(* Logix 5000 project; controller R5_CSS vendor 1 type 14 code 74 rev 19.11; software revision 19.01; part 4 of 20 *)
(* tags used below, declared in another part *)
   AlarmMaster : DINT;
   Coal_Tank_Heel_Inches : REAL;
   Coal_Tank_Height_Inches : REAL;
   FC101 : FLOW_CONTROL;   // QUENCH BASIN FLOW TRANSMITTER CONTROL
   FC108 : FLOW_CONTROL;   // QUENCH FEED FLOW TRANSMITTER
   FC140A : FLOW_CONTROL;   // QUENCH TOWER UPPER SPRAY FLOW CONTROL
   FC140B : FLOW_CONTROL;   // QUENCH TOWER LOWER SPRAY FLOW CONTROL
   FC403 : FLOW_CONTROL;   // COALESCER FLOW CONTROLLER FEEDS TCV108
   FCV410_LT_Hold : BOOL;
   FlowControlForce : BOOL;
   FlowControlForceONS : BOOL;
   FT101_SCP : SCLP;   // QUENCH BASIN FLOW TRANSMITTER SCALER
   FT108_SCP : SCLP;   // QUENCH FEED FLOW TRANSMITTER SCALER
   FT140A_SCP : SCLP;   // QUENCH TOWER UPPER SPRAY FIT SCALER
   FT140ABFlowMeterFailed : BOOL;
   FT140B_SCP : SCLP;   // QUENCH TOWER LOWER SPRAY FLOW TRANSMITTER SCALER
   FT403_SCP : SCLP;   // QUENCH CONDITIONING QUENCH WATER PHASE FLOW SCALER
   HART1 : HARTModuleDef;
   HARTData1 : HARTData;
   HEART_DATA : INT[122];
   LC101 : LEVEL_CONTROL;   // QUENCH TOWER BASIN LIT
   LC101_LT_Temp : REAL;
   LC303A : LEVEL_CONTROL;   // AQUEOUS PHASE OF PRIMARY SETTLER
   LC303A_LT_Raw : REAL;
   LC303B : LEVEL_CONTROL;   // INTERFACE LEVEL OF PRIMARY CONDENSER
   LC303B_LT_Raw : REAL;
   LC304 : LEVEL_CONTROL;   // SETTLER SECONDARY TANK INTERFACE LEVEL
   LC304_LT_Raw : REAL;
   LevelControlForce : BOOL;
   LevelControlForceONS : BOOL;
   LossOfSignal_mA : DINT;
   LT101_SCP : SCLP;   // QUENCH TOWER BASIN LIT SCALER
   LT303_Probe_Length_Inches : REAL;
   LT303_RAW : REAL[5];   // LT 303 RAW
   LT303_Scale_Param : REAL;
   LT304_SCP : SCLP;   // QUENCH COALESCING SEPARATOR SECONDARY CHAMBER LEVEL SCALER
   PC132 : PRESSURE_CONTROL;
   PC132_SCP : SCLP;
   PC133 : PRESSURE_CONTROL;
   PC133_SCP : SCLP;
   PC134 : PRESSURE_CONTROL;
   PC134_SCP : SCLP;
   PC408 : PRESSURE_CONTROL;
   PDT408_SCP : SCLP;
   QuenchFlowAutoControl : BOOL;
   QuenchFlowAutoControlPB : BOOL;
   QuenchFlowAutoControlPB_ONS : BOOL;
   QuenchFlowMeterFailed : BOOL;
   QuenchFlowMeterFailedTOF : TIMER;
   TC101A : TEMP_CONTROL;   // QUENCH BASIN TRANSFER BASIN A TEMPERATURE CONTROL
   TC101B : TEMP_CONTROL;   // QUENCH BASIN TRANSFER BASIN B TEMPERATURE CONTROL
   TC110 : TEMP_CONTROL;   // Quench Water Cartridge Heater Bundle Temp
   TC110_SCP : SCLP;
   TC112 : TEMP_CONTROL;   // Quench Water Cartridge Heater ProcessTemp
   TC112_SCP : SCLP;
   TC114A : TEMP_CONTROL;   // QUENCH BASIN SHELL TEMPERATURE CONTROL
   TC114B : TEMP_CONTROL;   // QUENCH BASIN LIQUID TEMPERATURE CONTROL
   TC123H : TEMP_CONTROL;
   TC123H_SCP : SCLP;
   TC135 : TEMP_CONTROL;
   TC135_SCP : SCLP;
   TC136 : TEMP_CONTROL;
   TC136_SCP : SCLP;
   TC137 : TEMP_CONTROL;
   TC137_SCP : SCLP;
   TC215 : TEMP_CONTROL;   // OVERHEAD CONDENSER CHILLED WATER TEMPERATURE TRANSMITTER CONTROL
   TC215_SCP : SCLP;   // OVERHEAD CONDENSER CHILLED WATER TEMPERATURE TRANSMITTER SCALER
   TC216 : TEMP_CONTROL;   // OVERHEAD CONDENSER BASIN TEMPERATURE CONTROL
   TC217 : TEMP_CONTROL;   // OVERHEAD CONDENSED CHILLED WATER RETURN TEMPERATURE CONTROL
   TC218 : TEMP_CONTROL;   // OVERHEAD CONDENSER CHILLED WATER SUPPLY TEMPERATURE CONTROL
   TC313A : TEMP_CONTROL;   // PRIMARY COALESCER SEPARATOR TEMPERATURE CONTROL
   TC313B : TEMP_CONTROL;   // PRIMARY COALESCER SHELL TEMPERATURE CONTROL
   TC319 : TEMP_CONTROL;   // COALESCER OIL CHAMBER PROCESS TEMPERATURE CONTROL
   TC320 : TEMP_CONTROL;   // COALESCER OIL CHAMBER SHELL TEMPERATURE TRANSMITTER CONTROL
   TC321A : TEMP_CONTROL;   // COALESCER OIL CHAMBER TRANSFER PUMP A TEMPERATURE TRANSMITTER
   TC321B : TEMP_CONTROL;   // COALESCER OIL CHAMBER TRANSFER PUMP B TEMPERATURE TRANSMITTER
   TC406 : TEMP_CONTROL;   // PROCESS WATER POST HX TEMPERATURE CONTROL
   TC406_SCP : SCLP;   // PROCESS WATER POST HX TEMPERATURE TRANSMITTER SCALER
   TC409 : TEMP_CONTROL;   // HX COOLING WATER SUPPLY TEMPERATURE CONTROL
   TC409_SCP : SCLP;   // HX COOLING WATER SUPPLY TEMPERATURE TRANSMITTER SCALER
   TC410 : TEMP_CONTROL;   // HX COOLING WATER RETURN TEMPERATURE CONTROL
   TC410_SCP : SCLP;   // HX COOLING WATER RETURN TEMPERATURE TRANSMITTER SCALER
   Test : INT[500];
   TT101A_SCP : SCLP;   // QUENCH BASIN TRANSFER BASIN A TEMPERATURE TRANSMITTER SCALER
   TT101B_SCP : SCLP;   // QUENCH BASIN TRANSFER BASIN B TEMPERATURE TRANSMITTER SCALER
   TT114A_SCP : SCLP;   // QUENCH BASIN SHELL TEMPERATURE TRANSMITTER SCALER
   TT114B_SCP : SCLP;   // QUENCH BASIN LIQUID TEMPERATURE TRANSMITTER SCALER
   TT216_SCP : SCLP;   // OVERHEAD CONDENSER BASIN TEMPERATURE TRANSMITTER SCALER
   TT217_SCP : SCLP;   // OVERHEAD CONDENSED CHILLED WATER RETURN TEMPERATURE TRANSMITTER
   TT218_SCP : SCLP;   // OVERHEAD CONDENSER CHILLED WATER SUPPLY TEMPERATURE SCALER
   TT313A_SCP : SCLP;   // PRIMARY COALESCER SEPARATOR TEMPERATURE TRANSMITTER SCALER
   TT313B_SCP : SCLP;   // PRIMARY COALESCER SHELL TEMPERATURE TRANSMITTER SCALER
   TT319_SCP : SCLP;   // COALESCER OIL CHAMBER SHELL TEMPERATURE TRANSMITTER SCALER
   TT320_SCP : SCLP;   // COALESCER OIL CHAMBER SHELL TEMPERATURE TRANSMITTER SCALER
   TT321A_SCP : SCLP;   // COALESCER OIL CHAMBER TRANSFER PUMP A TEMPERATURE TRANSMITTER SCALER
   TT321B_SCP : SCLP;   // COALESCER OIL CHAMBER TRANSFER PUMP B TEMPERATURE TRANSMITTER
(* MainProgram, continued *)

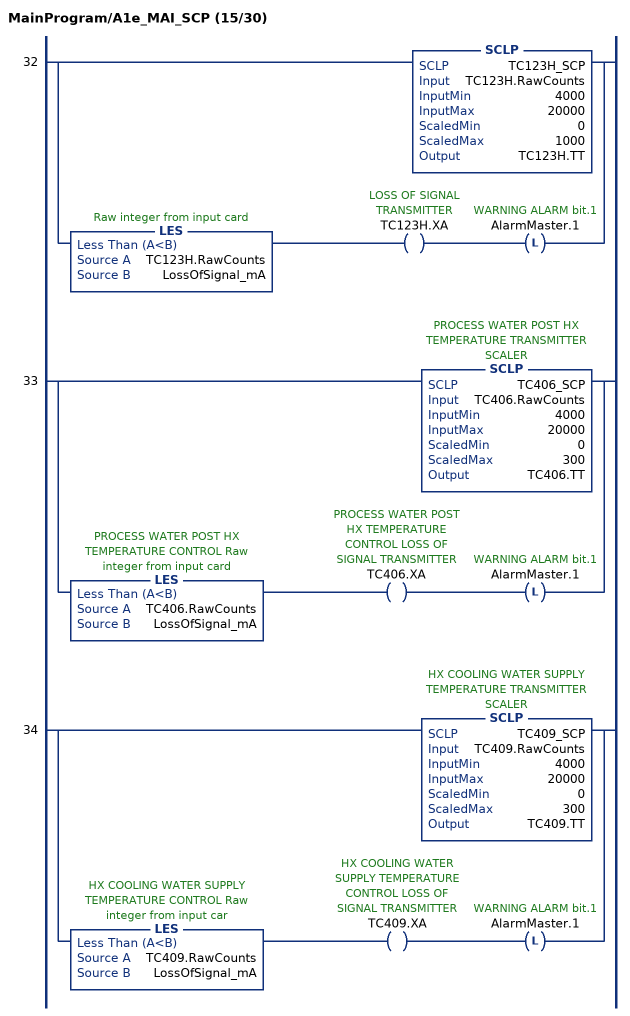
   [picture p58: MainProgram/A1e_MAI_SCP rungs 32-34]
   32: [SCLP(TC123H_SCP,TC123H.RawCounts,4000,20000,0,1000,TC123H.TT) ,LES(TC123H.RawCounts,LossOfSignal_mA) OTE(TC123H.XA) OTL(AlarmMaster.1) ];
   33: [SCLP(TC406_SCP,TC406.RawCounts,4000,20000,0,300,TC406.TT) ,LES(TC406.RawCounts,LossOfSignal_mA) OTE(TC406.XA) OTL(AlarmMaster.1) ];
   34: [SCLP(TC409_SCP,TC409.RawCounts,4000,20000,0,300,TC409.TT) ,LES(TC409.RawCounts,LossOfSignal_mA) OTE(TC409.XA) OTL(AlarmMaster.1) ];
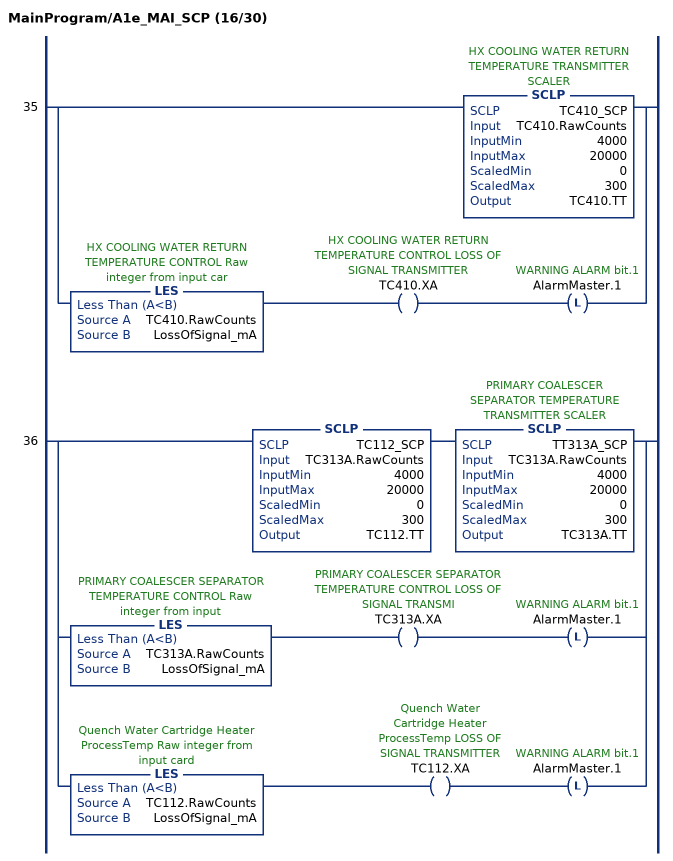
   35: [SCLP(TC410_SCP,TC410.RawCounts,4000,20000,0,300,TC410.TT) ,LES(TC410.RawCounts,LossOfSignal_mA) OTE(TC410.XA) OTL(AlarmMaster.1) ];
   36: [SCLP(TC112_SCP,TC313A.RawCounts,4000,20000,0,300,TC112.TT) SCLP(TT313A_SCP,TC313A.RawCounts,4000,20000,0,300,TC313A.TT) ,LES(TC313A.RawCounts,LossOfSignal_mA) OTE(TC313A.XA) OTL(AlarmMaster.1) ,LES(TC112.RawCounts,LossOfSignal_mA) OTE(TC112.XA) OTL(AlarmMaster.1) ];
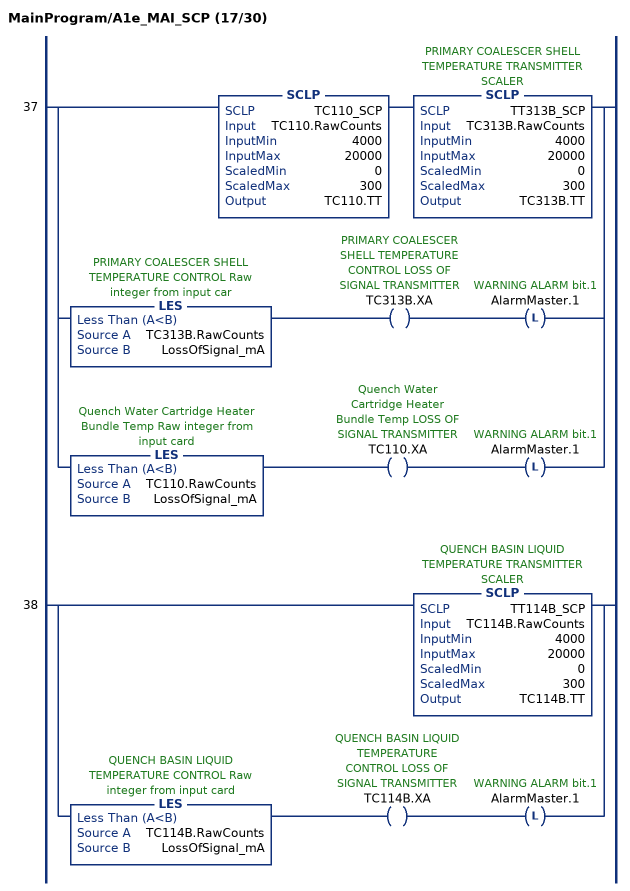
   37: [SCLP(TC110_SCP,TC110.RawCounts,4000,20000,0,300,TC110.TT) SCLP(TT313B_SCP,TC313B.RawCounts,4000,20000,0,300,TC313B.TT) ,LES(TC313B.RawCounts,LossOfSignal_mA) OTE(TC313B.XA) OTL(AlarmMaster.1) ,LES(TC110.RawCounts,LossOfSignal_mA) OTE(TC110.XA) OTL(AlarmMaster.1) ];
   38: [SCLP(TT114B_SCP,TC114B.RawCounts,4000,20000,0,300,TC114B.TT) ,LES(TC114B.RawCounts,LossOfSignal_mA) OTE(TC114B.XA) OTL(AlarmMaster.1) ];
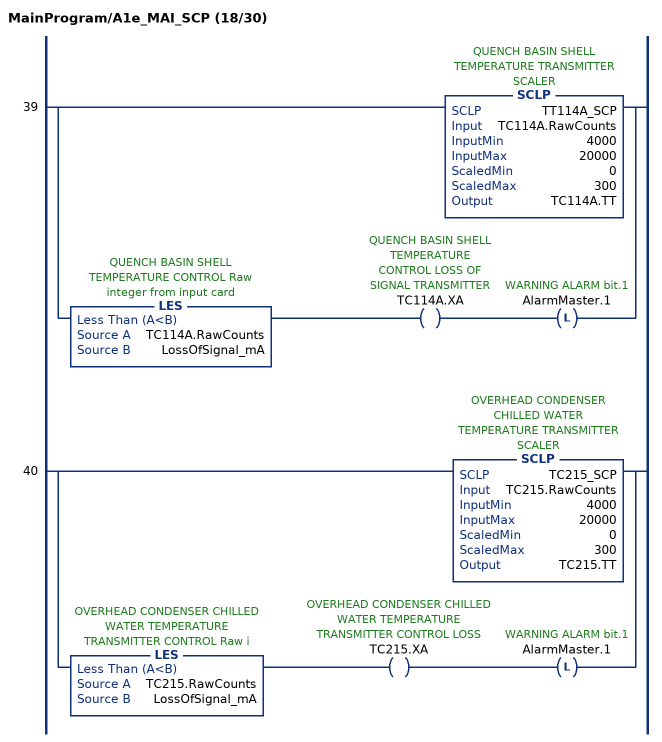
   39: [SCLP(TT114A_SCP,TC114A.RawCounts,4000,20000,0,300,TC114A.TT) ,LES(TC114A.RawCounts,LossOfSignal_mA) OTE(TC114A.XA) OTL(AlarmMaster.1) ];
   40: [SCLP(TC215_SCP,TC215.RawCounts,4000,20000,0,300,TC215.TT) ,LES(TC215.RawCounts,LossOfSignal_mA) OTE(TC215.XA) OTL(AlarmMaster.1) ];
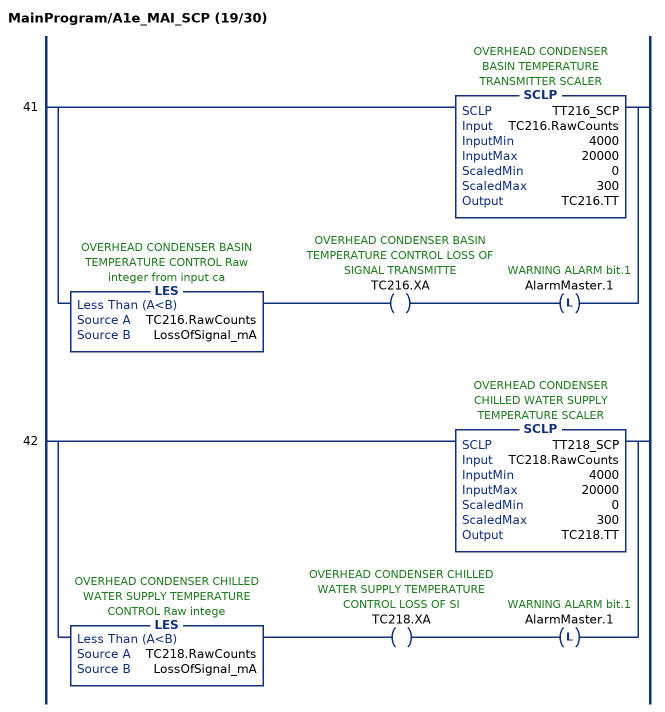
   41: [SCLP(TT216_SCP,TC216.RawCounts,4000,20000,0,300,TC216.TT) ,LES(TC216.RawCounts,LossOfSignal_mA) OTE(TC216.XA) OTL(AlarmMaster.1) ];
   42: [SCLP(TT218_SCP,TC218.RawCounts,4000,20000,0,300,TC218.TT) ,LES(TC218.RawCounts,LossOfSignal_mA) OTE(TC218.XA) OTL(AlarmMaster.1) ];
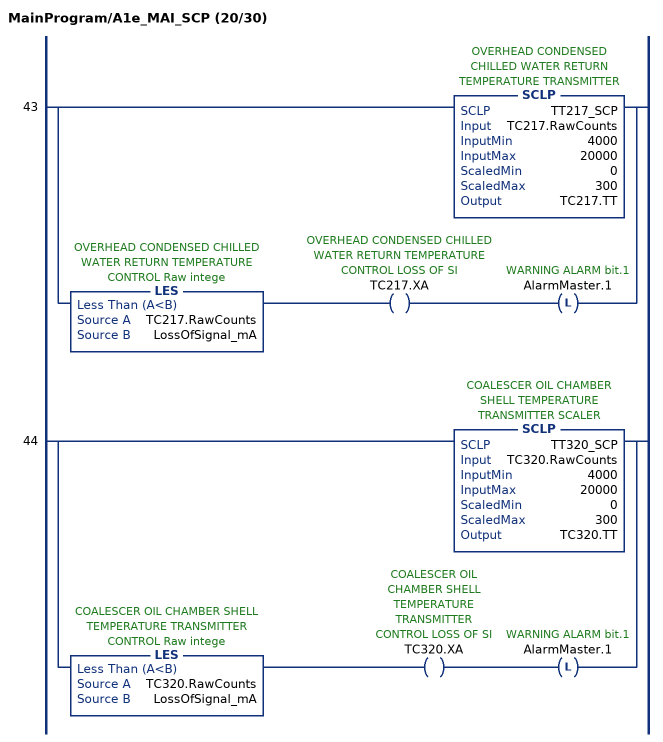
   43: [SCLP(TT217_SCP,TC217.RawCounts,4000,20000,0,300,TC217.TT) ,LES(TC217.RawCounts,LossOfSignal_mA) OTE(TC217.XA) OTL(AlarmMaster.1) ];
   44: [SCLP(TT320_SCP,TC320.RawCounts,4000,20000,0,300,TC320.TT) ,LES(TC320.RawCounts,LossOfSignal_mA) OTE(TC320.XA) OTL(AlarmMaster.1) ];
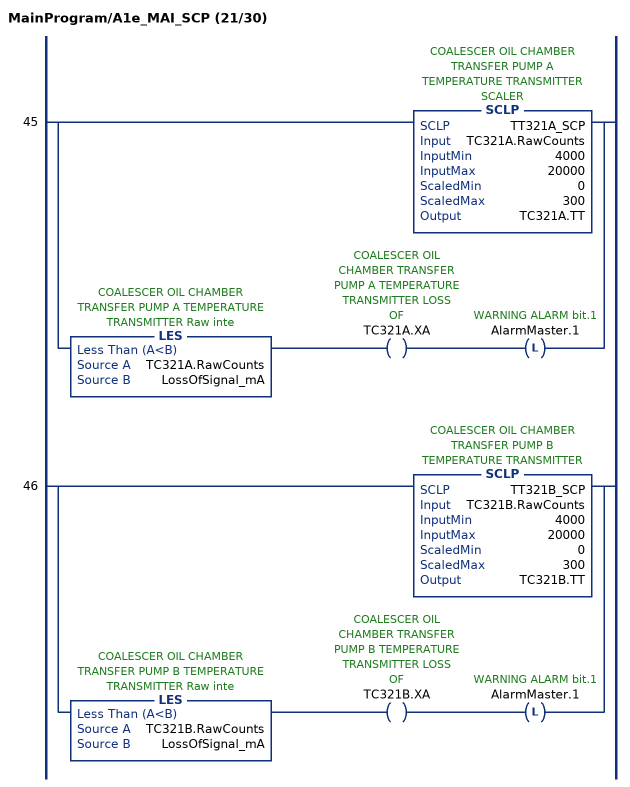
   45: [SCLP(TT321A_SCP,TC321A.RawCounts,4000,20000,0,300,TC321A.TT) ,LES(TC321A.RawCounts,LossOfSignal_mA) OTE(TC321A.XA) OTL(AlarmMaster.1) ];
   46: [SCLP(TT321B_SCP,TC321B.RawCounts,4000,20000,0,300,TC321B.TT) ,LES(TC321B.RawCounts,LossOfSignal_mA) OTE(TC321B.XA) OTL(AlarmMaster.1) ];
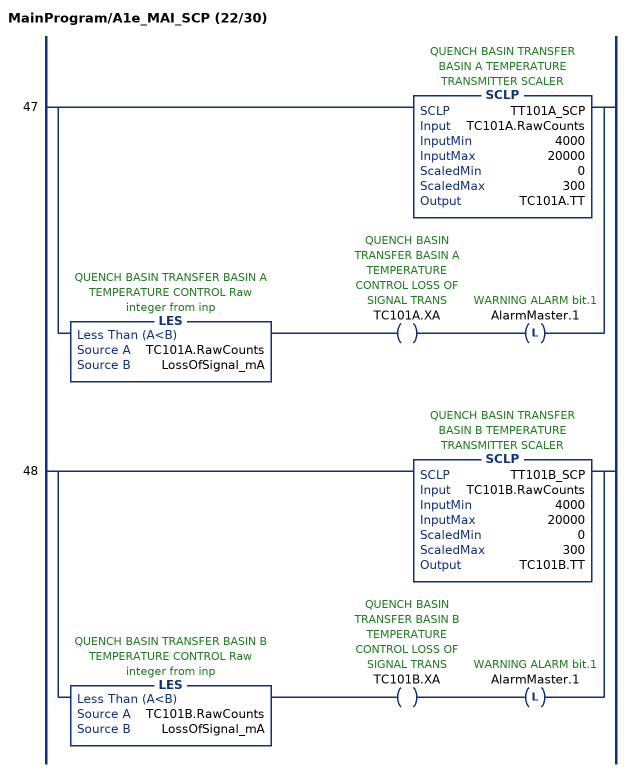
   47: [SCLP(TT101A_SCP,TC101A.RawCounts,4000,20000,0,300,TC101A.TT) ,LES(TC101A.RawCounts,LossOfSignal_mA) OTE(TC101A.XA) OTL(AlarmMaster.1) ];
   48: [SCLP(TT101B_SCP,TC101B.RawCounts,4000,20000,0,300,TC101B.TT) ,LES(TC101B.RawCounts,LossOfSignal_mA) OTE(TC101B.XA) OTL(AlarmMaster.1) ];
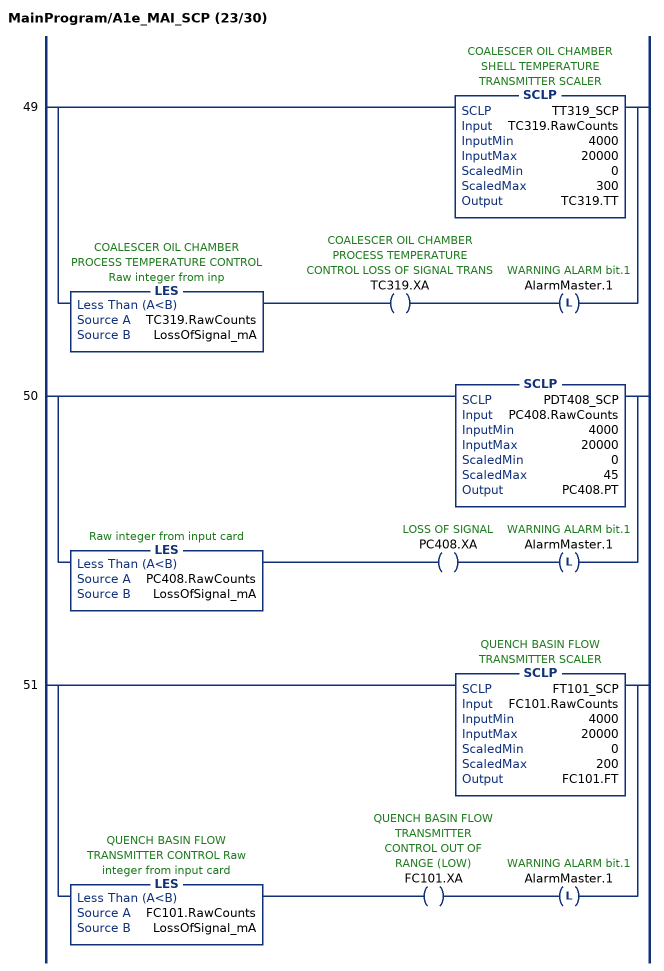
   49: [SCLP(TT319_SCP,TC319.RawCounts,4000,20000,0,300,TC319.TT) ,LES(TC319.RawCounts,LossOfSignal_mA) OTE(TC319.XA) OTL(AlarmMaster.1) ];
   50: [SCLP(PDT408_SCP,PC408.RawCounts,4000,20000,0,45,PC408.PT) ,LES(PC408.RawCounts,LossOfSignal_mA) OTE(PC408.XA) OTL(AlarmMaster.1) ];
   51: [SCLP(FT101_SCP,FC101.RawCounts,4000,20000,0,200,FC101.FT) ,LES(FC101.RawCounts,LossOfSignal_mA) OTE(FC101.XA) OTL(AlarmMaster.1) ];
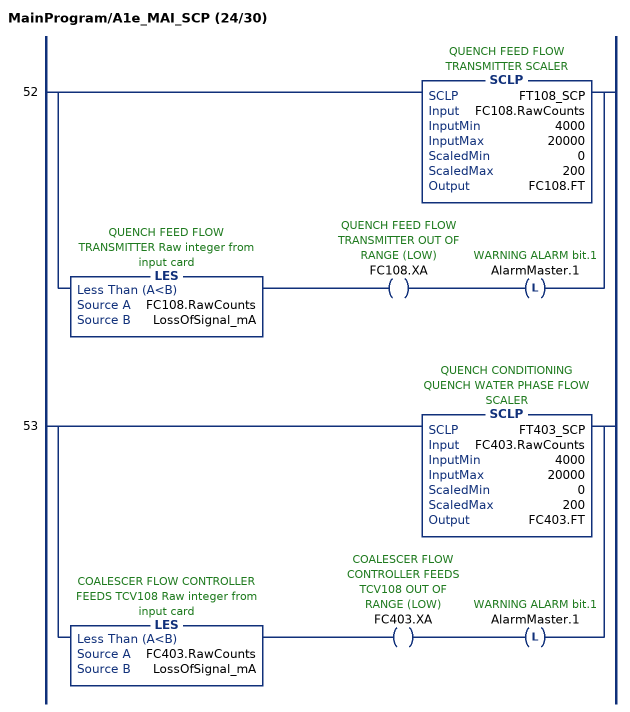
   52: [SCLP(FT108_SCP,FC108.RawCounts,4000,20000,0,200,FC108.FT) ,LES(FC108.RawCounts,LossOfSignal_mA) OTE(FC108.XA) OTL(AlarmMaster.1) ];
   53: [SCLP(FT403_SCP,FC403.RawCounts,4000,20000,0,200,FC403.FT) ,LES(FC403.RawCounts,LossOfSignal_mA) OTE(FC403.XA) OTL(AlarmMaster.1) ];
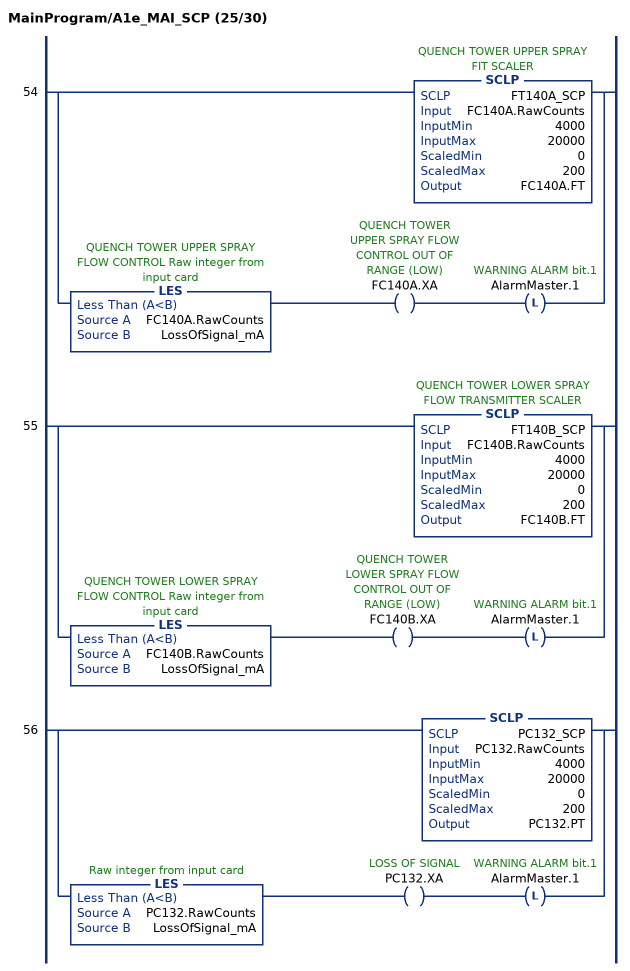
   54: [SCLP(FT140A_SCP,FC140A.RawCounts,4000,20000,0,200,FC140A.FT) ,LES(FC140A.RawCounts,LossOfSignal_mA) OTE(FC140A.XA) OTL(AlarmMaster.1) ];
   55: [SCLP(FT140B_SCP,FC140B.RawCounts,4000,20000,0,200,FC140B.FT) ,LES(FC140B.RawCounts,LossOfSignal_mA) OTE(FC140B.XA) OTL(AlarmMaster.1) ];
   56: [SCLP(PC132_SCP,PC132.RawCounts,4000,20000,0,200,PC132.PT) ,LES(PC132.RawCounts,LossOfSignal_mA) OTE(PC132.XA) OTL(AlarmMaster.1) ];
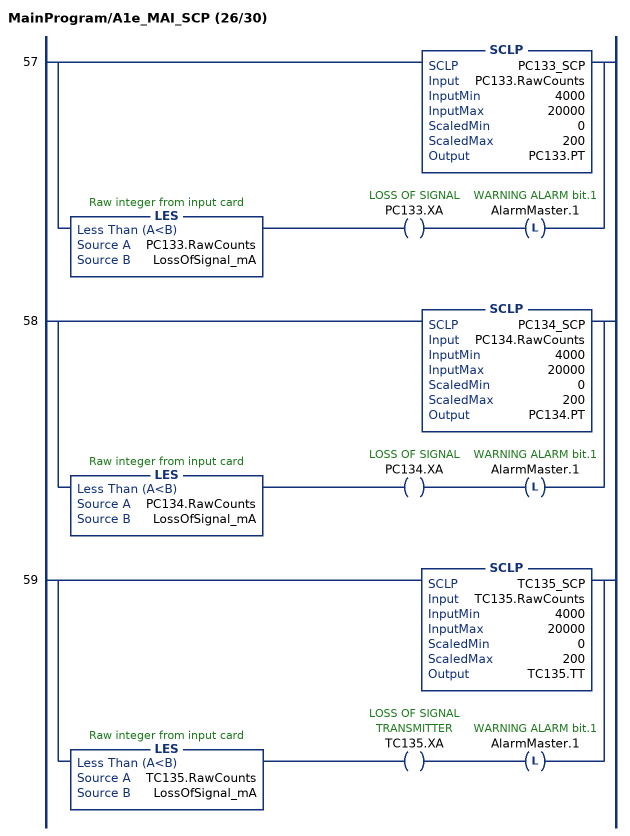
   57: [SCLP(PC133_SCP,PC133.RawCounts,4000,20000,0,200,PC133.PT) ,LES(PC133.RawCounts,LossOfSignal_mA) OTE(PC133.XA) OTL(AlarmMaster.1) ];
   58: [SCLP(PC134_SCP,PC134.RawCounts,4000,20000,0,200,PC134.PT) ,LES(PC134.RawCounts,LossOfSignal_mA) OTE(PC134.XA) OTL(AlarmMaster.1) ];
   59: [SCLP(TC135_SCP,TC135.RawCounts,4000,20000,0,200,TC135.TT) ,LES(TC135.RawCounts,LossOfSignal_mA) OTE(TC135.XA) OTL(AlarmMaster.1) ];
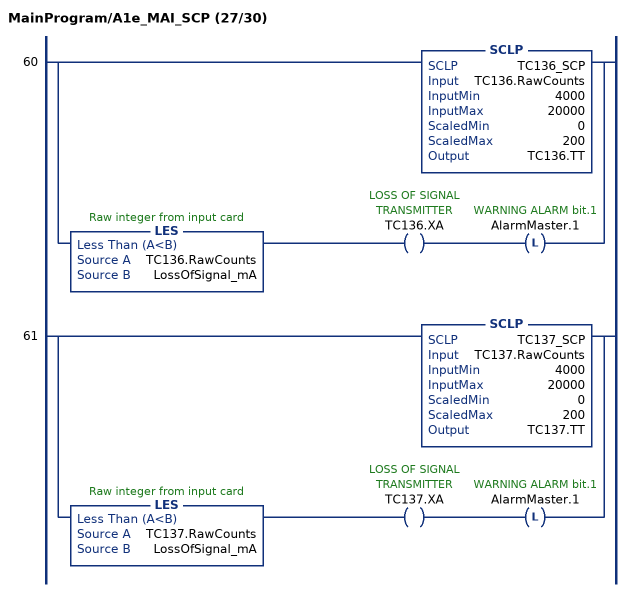
   60: [SCLP(TC136_SCP,TC136.RawCounts,4000,20000,0,200,TC136.TT) ,LES(TC136.RawCounts,LossOfSignal_mA) OTE(TC136.XA) OTL(AlarmMaster.1) ];
   61: [SCLP(TC137_SCP,TC137.RawCounts,4000,20000,0,200,TC137.TT) ,LES(TC137.RawCounts,LossOfSignal_mA) OTE(TC137.XA) OTL(AlarmMaster.1) ];
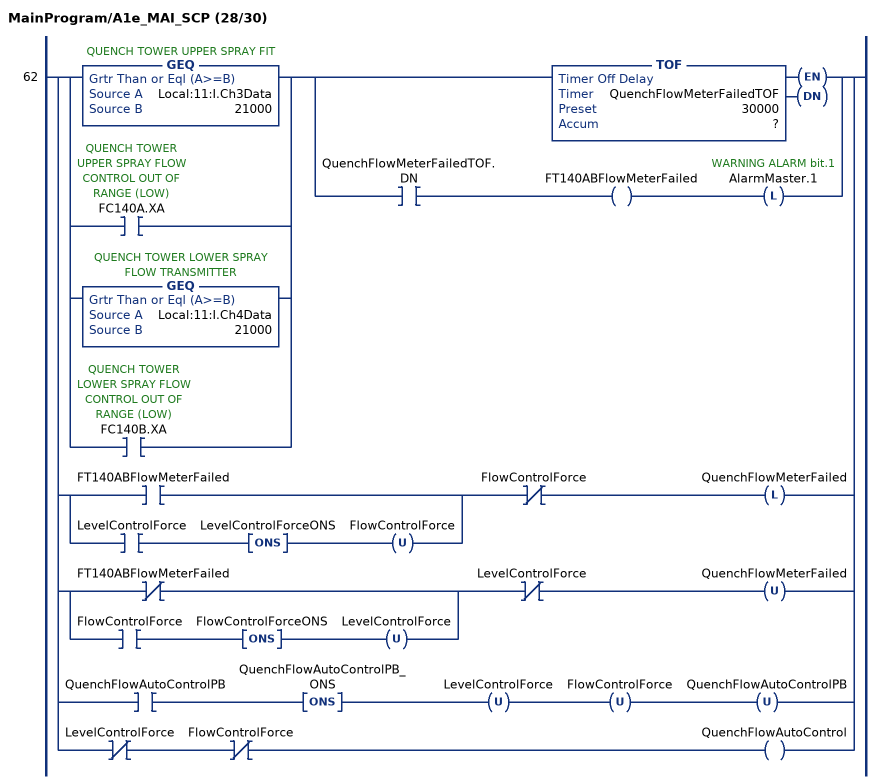
   62: [[GEQ(Local:11:I.Ch3Data,21000) ,XIC(FC140A.XA) ,GEQ(Local:11:I.Ch4Data,21000) ,XIC(FC140B.XA) ] [TOF(QuenchFlowMeterFailedTOF,?,?) ,XIC(QuenchFlowMeterFailedTOF.DN) OTE(FT140ABFlowMeterFailed) OTL(AlarmMaster.1) ] ,[XIC(FT140ABFlowMeterFailed) ,XIC(LevelControlForce) ONS(LevelControlForceONS) OTU(FlowControlForce) ] XIO(FlowControlForce) OTL(QuenchFlowMeterFailed) ,[XIO(FT140ABFlowMeterFailed) ,XIC(FlowControlForce) ONS(FlowControlForceONS) OTU(LevelControlForce) ] XIO(LevelControlForce) OTU(QuenchFlowMeterFailed) ,XIC(QuenchFlowAutoControlPB) ONS(QuenchFlowAutoControlPB_ONS) OTU(LevelControlForce) OTU(FlowControlForce) OTU(QuenchFlowAutoControlPB) ,XIO(LevelControlForce) XIO(FlowControlForce) OTE(QuenchFlowAutoControl) ];
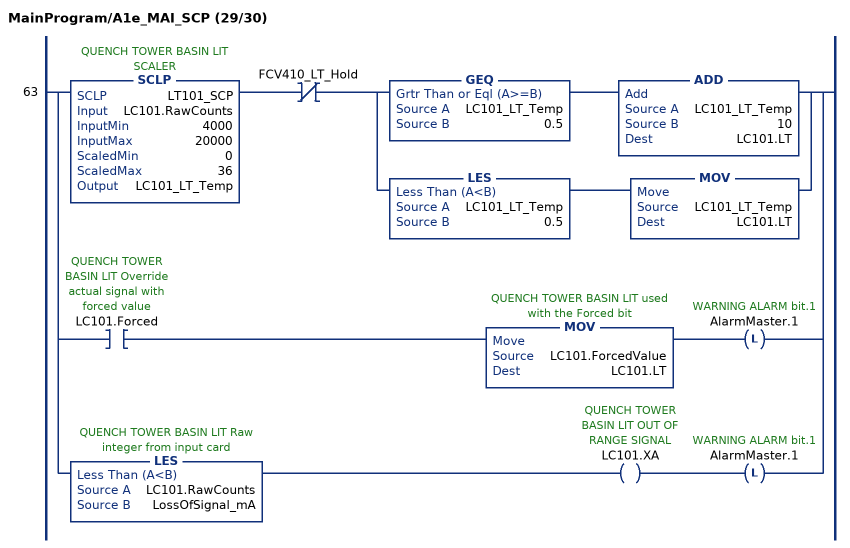
   63: [SCLP(LT101_SCP,LC101.RawCounts,4000,20000,0,36,LC101_LT_Temp) XIO(FCV410_LT_Hold) [GEQ(LC101_LT_Temp,0.5) ADD(LC101_LT_Temp,10,LC101.LT) ,LES(LC101_LT_Temp,0.5) MOV(LC101_LT_Temp,LC101.LT) ] ,XIC(LC101.Forced) MOV(LC101.ForcedValue,LC101.LT) OTL(AlarmMaster.1) ,LES(LC101.RawCounts,LossOfSignal_mA) OTE(LC101.XA) OTL(AlarmMaster.1) ];
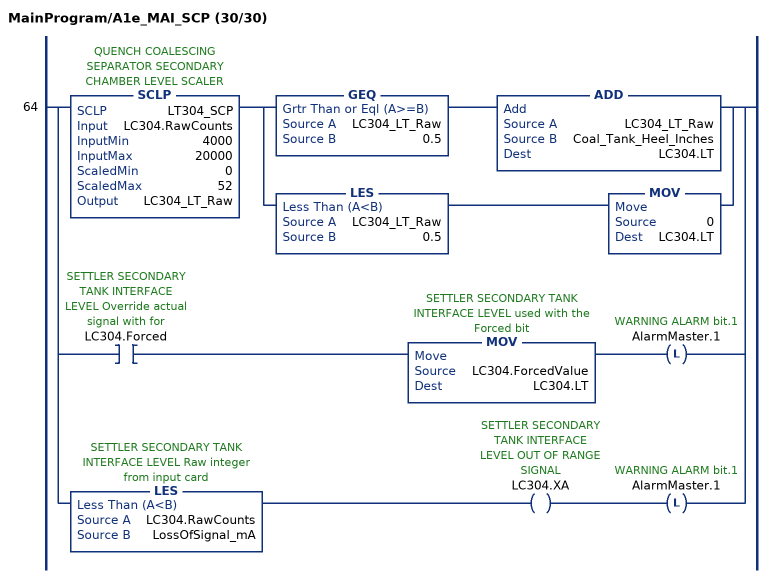
   64: [SCLP(LT304_SCP,LC304.RawCounts,4000,20000,0,52,LC304_LT_Raw) [GEQ(LC304_LT_Raw,0.5) ADD(LC304_LT_Raw,Coal_Tank_Heel_Inches,LC304.LT) ,LES(LC304_LT_Raw,0.5) MOV(0,LC304.LT) ] ,XIC(LC304.Forced) MOV(LC304.ForcedValue,LC304.LT) OTL(AlarmMaster.1) ,LES(LC304.RawCounts,LossOfSignal_mA) OTE(LC304.XA) OTL(AlarmMaster.1) ];
END_ROUTINE

ROUTINE A2a_MM_HART   (* ladder *)
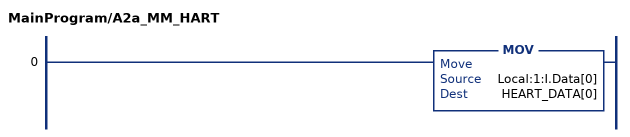
   0: MOV(Local:1:I.Data[0],HEART_DATA[0]);
END_ROUTINE

ROUTINE A2b_HART_READ   (* ladder *)
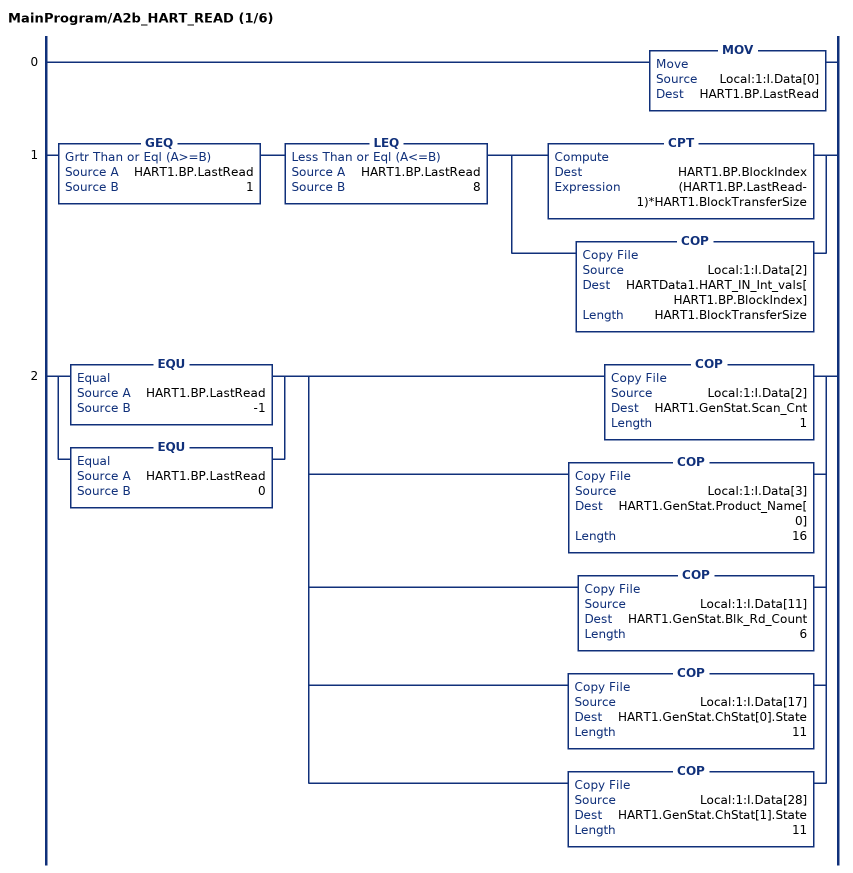
   0: MOV(Local:1:I.Data[0],HART1.BP.LastRead);
   1: GEQ(HART1.BP.LastRead,1)LEQ(HART1.BP.LastRead,8)[CPT(HART1.BP.BlockIndex,(HART1.BP.LastRead-1)*HART1.BlockTransferSize) ,COP(Local:1:I.Data[2],HARTData1.HART_IN_Int_vals[HART1.BP.BlockIndex],HART1.BlockTransferSize) ];
   2: [EQU(HART1.BP.LastRead,-1) ,EQU(HART1.BP.LastRead,0) ][COP(Local:1:I.Data[2],HART1.GenStat.Scan_Cnt,1) ,COP(Local:1:I.Data[3],HART1.GenStat.Product_Name[0],16) ,COP(Local:1:I.Data[11],HART1.GenStat.Blk_Rd_Count,6) ,COP(Local:1:I.Data[17],HART1.GenStat.ChStat[0].State,11) ,COP(Local:1:I.Data[28],HART1.GenStat.ChStat[1].State,11) ];
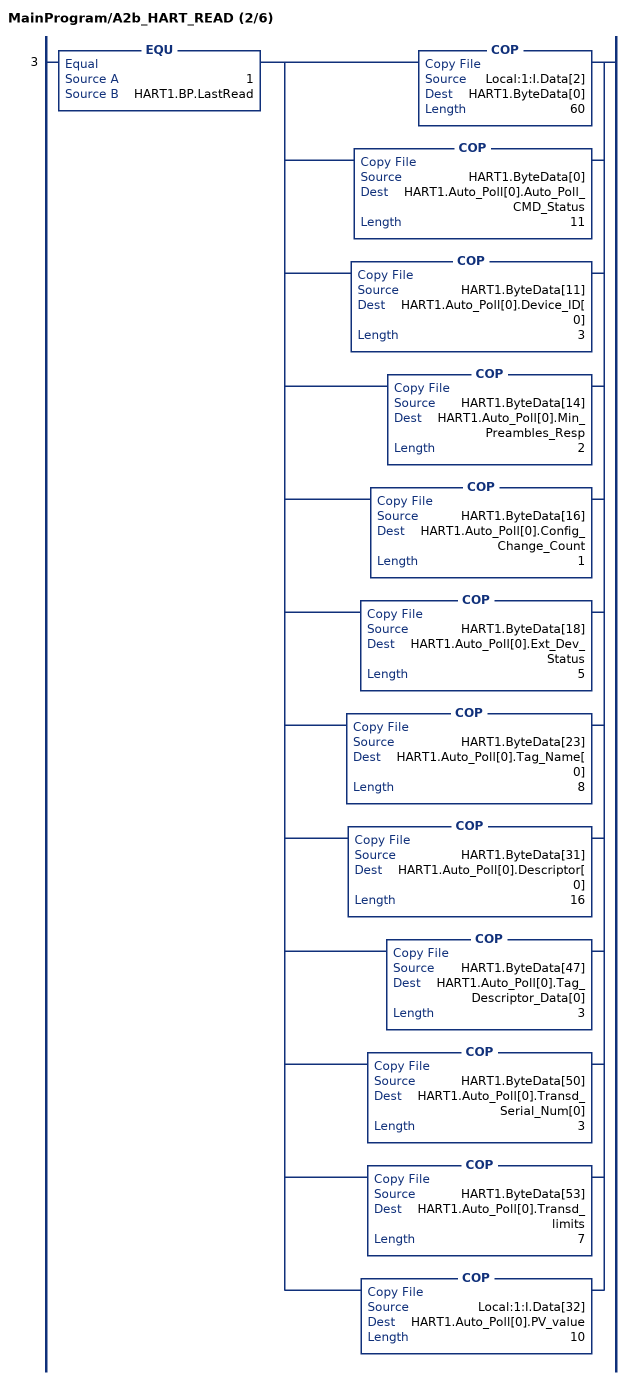
   3: EQU(1,HART1.BP.LastRead)[COP(Local:1:I.Data[2],HART1.ByteData[0],60) ,COP(HART1.ByteData[0],HART1.Auto_Poll[0].Auto_Poll_CMD_Status,11) ,COP(HART1.ByteData[11],HART1.Auto_Poll[0].Device_ID[0],3) ,COP(HART1.ByteData[14],HART1.Auto_Poll[0].Min_Preambles_Resp,2) ,COP(HART1.ByteData[16],HART1.Auto_Poll[0].Config_Change_Count,1) ,COP(HART1.ByteData[18],HART1.Auto_Poll[0].Ext_Dev_Status,5) ,COP(HART1.ByteData[23],HART1.Auto_Poll[0].Tag_Name[0],8) ,COP(HART1.ByteData[31],HART1.Auto_Poll[0].Descriptor[0],16) ,COP(HART1.ByteData[47],HART1.Auto_Poll[0].Tag_Descriptor_Data[0],3) ,COP(HART1.ByteData[50],HART1.Auto_Poll[0].Transd_Serial_Num[0],3) ,COP(HART1.ByteData[53],HART1.Auto_Poll[0].Transd_limits,7) ,COP(Local:1:I.Data[32],HART1.Auto_Poll[0].PV_value,10) ];
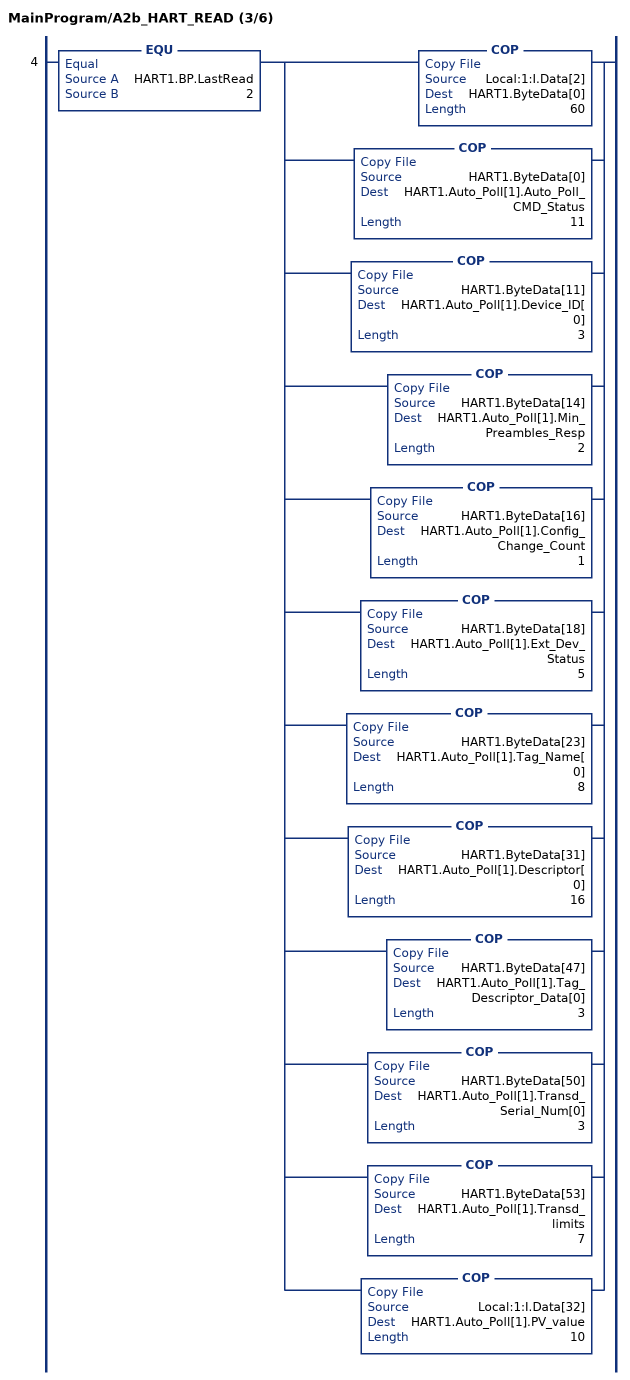
   4: EQU(HART1.BP.LastRead,2)[COP(Local:1:I.Data[2],HART1.ByteData[0],60) ,COP(HART1.ByteData[0],HART1.Auto_Poll[1].Auto_Poll_CMD_Status,11) ,COP(HART1.ByteData[11],HART1.Auto_Poll[1].Device_ID[0],3) ,COP(HART1.ByteData[14],HART1.Auto_Poll[1].Min_Preambles_Resp,2) ,COP(HART1.ByteData[16],HART1.Auto_Poll[1].Config_Change_Count,1) ,COP(HART1.ByteData[18],HART1.Auto_Poll[1].Ext_Dev_Status,5) ,COP(HART1.ByteData[23],HART1.Auto_Poll[1].Tag_Name[0],8) ,COP(HART1.ByteData[31],HART1.Auto_Poll[1].Descriptor[0],16) ,COP(HART1.ByteData[47],HART1.Auto_Poll[1].Tag_Descriptor_Data[0],3) ,COP(HART1.ByteData[50],HART1.Auto_Poll[1].Transd_Serial_Num[0],3) ,COP(HART1.ByteData[53],HART1.Auto_Poll[1].Transd_limits,7) ,COP(Local:1:I.Data[32],HART1.Auto_Poll[1].PV_value,10) ];
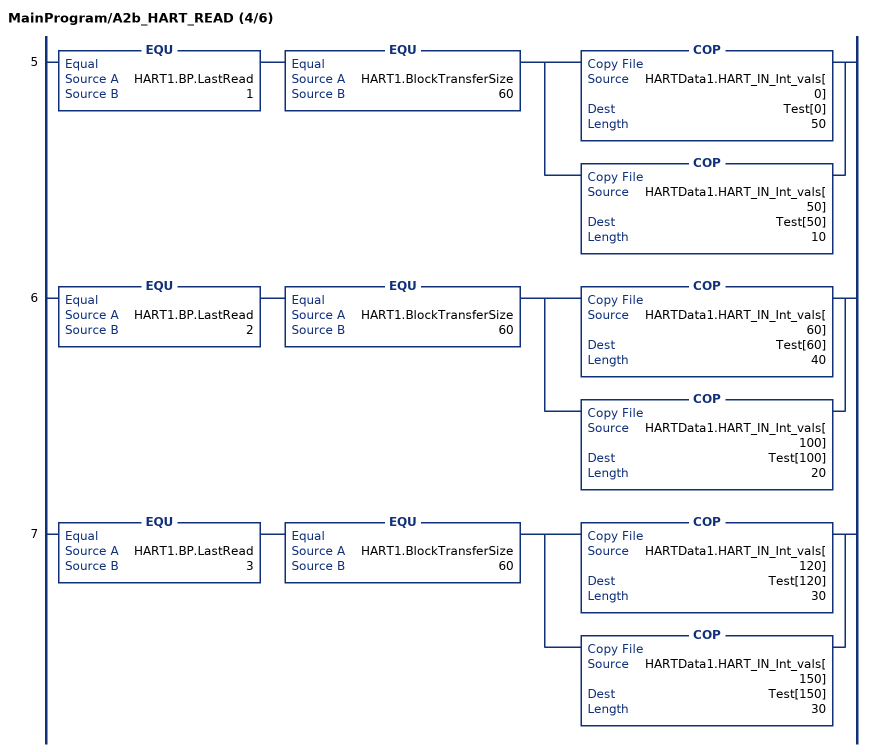
   5: EQU(HART1.BP.LastRead,1)EQU(HART1.BlockTransferSize,60)[COP(HARTData1.HART_IN_Int_vals[0],Test[0],50) ,COP(HARTData1.HART_IN_Int_vals[50],Test[50],10) ];
   6: EQU(HART1.BP.LastRead,2)EQU(HART1.BlockTransferSize,60)[COP(HARTData1.HART_IN_Int_vals[60],Test[60],40) ,COP(HARTData1.HART_IN_Int_vals[100],Test[100],20) ];
   7: EQU(HART1.BP.LastRead,3)EQU(HART1.BlockTransferSize,60)[COP(HARTData1.HART_IN_Int_vals[120],Test[120],30) ,COP(HARTData1.HART_IN_Int_vals[150],Test[150],30) ];
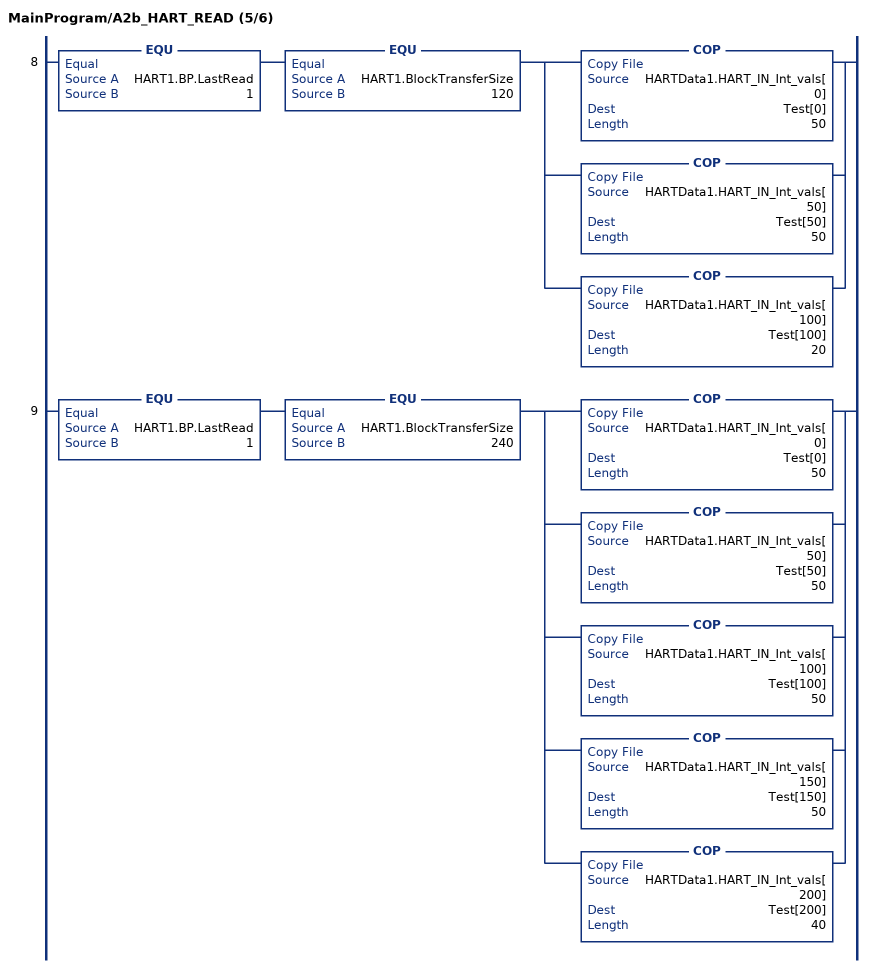
   8: EQU(HART1.BP.LastRead,1)EQU(HART1.BlockTransferSize,120)[COP(HARTData1.HART_IN_Int_vals[0],Test[0],50) ,COP(HARTData1.HART_IN_Int_vals[50],Test[50],50) ,COP(HARTData1.HART_IN_Int_vals[100],Test[100],20) ];
   9: EQU(HART1.BP.LastRead,1)EQU(HART1.BlockTransferSize,240)[COP(HARTData1.HART_IN_Int_vals[0],Test[0],50) ,COP(HARTData1.HART_IN_Int_vals[50],Test[50],50) ,COP(HARTData1.HART_IN_Int_vals[100],Test[100],50) ,COP(HARTData1.HART_IN_Int_vals[150],Test[150],50) ,COP(HARTData1.HART_IN_Int_vals[200],Test[200],40) ];
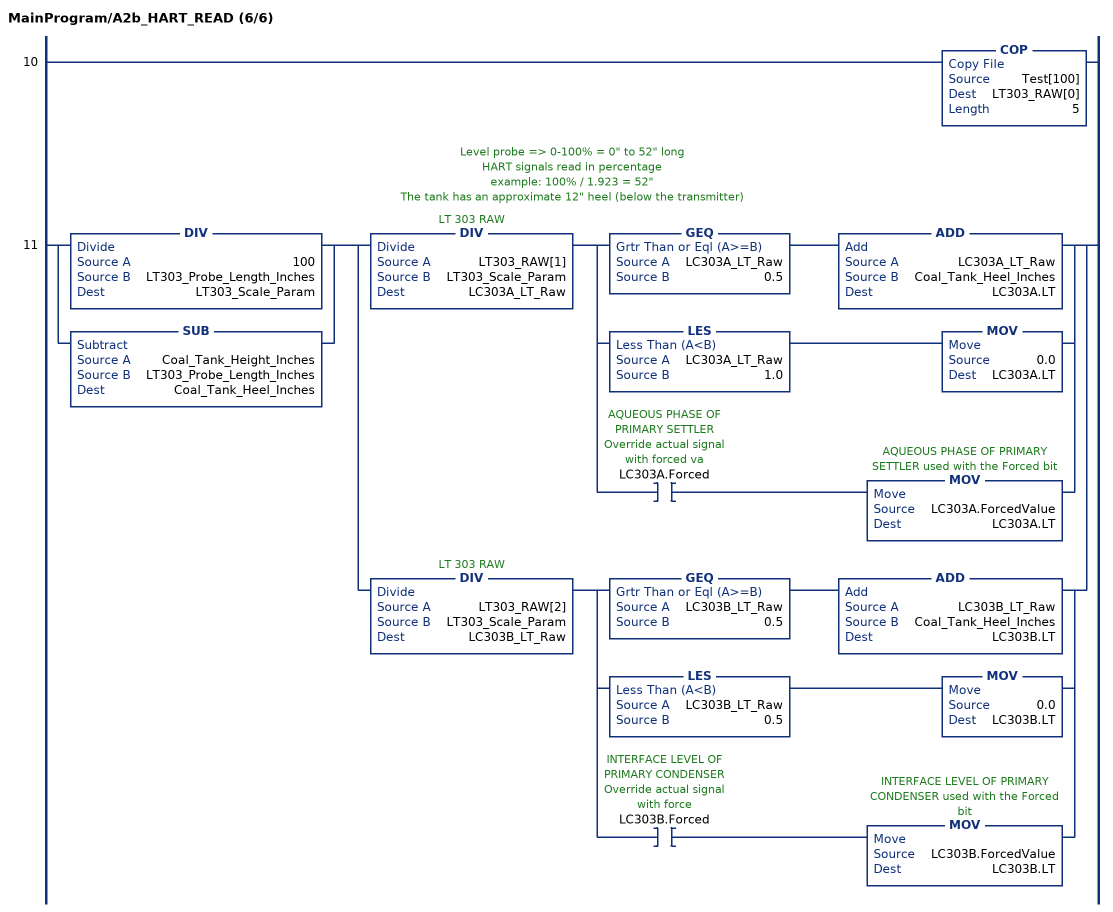
   10: COP(Test[100],LT303_RAW[0],5);
   // Level probe => 0-100% = 0" to 52" long
   // HART signals read in percentage
   // example: 100% / 1.923 = 52"
   // The tank has an approximate 12" heel (below the transmitter)
   11: [DIV(100,LT303_Probe_Length_Inches,LT303_Scale_Param) ,SUB(Coal_Tank_Height_Inches,LT303_Probe_Length_Inches,Coal_Tank_Heel_Inches) ][DIV(LT303_RAW[1],LT303_Scale_Param,LC303A_LT_Raw) [GEQ(LC303A_LT_Raw,0.5) ADD(LC303A_LT_Raw,Coal_Tank_Heel_Inches,LC303A.LT) ,LES(LC303A_LT_Raw,1.0) MOV(0.0,LC303A.LT) ,XIC(LC303A.Forced) MOV(LC303A.ForcedValue,LC303A.LT) ] ,DIV(LT303_RAW[2],LT303_Scale_Param,LC303B_LT_Raw) [GEQ(LC303B_LT_Raw,0.5) ADD(LC303B_LT_Raw,Coal_Tank_Heel_Inches,LC303B.LT) ,LES(LC303B_LT_Raw,0.5) MOV(0.0,LC303B.LT) ,XIC(LC303B.Forced) MOV(LC303B.ForcedValue,LC303B.LT) ] ];
END_ROUTINE
